stXStage.bLimitForwardEnable := TRUE;
stXStage.bLimitBackwardEnable := TRUE;
stXStage.bHardwareEnable := TRUE;
stXStage.bPowerSelf := TRUE;

fbYStage(stMotionStage:=stYStage);
fbXStage(stMotionStage:=stXStage);

// We need to update from PLC or from EPICS, but not both
fbArrCheckWrite(
    astPositionState:=astPositionState,
    bCheck:=TRUE,
    bSave:=FALSE,
);
IF NOT fbArrCheckWrite.bHadWrite THEN
    astPositionState[ENUM_TM2K4_States.OUT] := stOut;
    astPositionState[ENUM_TM2K4_States.TARGET1a] := stTarget1a;
    astPositionState[ENUM_TM2K4_States.TARGET1b] := stTarget1b;
    astPositionState[ENUM_TM2K4_States.TARGET2a] := stTarget2a;
    astPositionState[ENUM_TM2K4_States.TARGET2b] := stTarget2b;
    astPositionState[ENUM_TM2K4_States.TARGET3a] := stTarget3a;
    astPositionState[ENUM_TM2K4_States.TARGET3b] := stTarget3b;
    astPositionState[ENUM_TM2K4_States.YAG] := stTarget4;
    astPositionState[ENUM_TM2K4_States.DIODE] := stTarget5;
END_IF

fbStates(
    stMotionStage:=stYStage,
    astPositionState:=astPositionState,
    eEnumSet:=eEnumSet,
    eEnumGet:=eEnumGet,
    fbFFHWO:=fbFFHWO,
    fbArbiter:=fbArbiter,
    bEnableMotion:=bEnableMotion,
    bEnableBeamParams:=bEnableBeamParams,
    bEnablePositionLimits:=bEnablePositionLimits,
    sDeviceName:=sDeviceName,
    sTransitionKey:=sTransitionKey,
    bReadDBNow:=bReadDBNow,
    stDbStateParams=>stDbStateParams,
);

fbArrCheckWrite(
    astPositionState:=astPositionState,
    bCheck:=FALSE,
    bSave:=TRUE,
);

stOut := astPositionState[ENUM_TM2K4_States.OUT];
stTarget1a := astPositionState[ENUM_TM2K4_States.TARGET1a];
stTarget1b := astPositionState[ENUM_TM2K4_States.TARGET1b];
stTarget2a := astPositionState[ENUM_TM2K4_States.TARGET2a];
stTarget2b := astPositionState[ENUM_TM2K4_States.TARGET2b];
stTarget3a := astPositionState[ENUM_TM2K4_States.TARGET3a];
stTarget3b := astPositionState[ENUM_TM2K4_States.TARGET3b];
stTarget4 := astPositionState[ENUM_TM2K4_States.YAG];
stTarget5 := astPositionState[ENUM_TM2K4_States.DIODE];

fbTempSensor1(
    fFaultThreshold:=fbStates.stDbStateParams.stReactiveParams.nTempSP,
    bVeto:=eEnumGet = ENUM_TM2K4_States.OUT,
    sDevName:=sDeviceName,
    io_fbFFHWO:=fbFFHWO,
);
fbFlowMeter();

END_FUNCTION_BLOCK

// ---- POUs/PRG_SP1K4.TcPOU
  PROGRAM PRG_SP1K4
VAR
    fbMotionLensX: FB_MotionStage;
    fbMotionFoilX: FB_MotionStage;
    fbMotionZPX: FB_MotionStage;
    fbMotionZPY: FB_MotionStage;
    fbMotionZPZ: FB_MotionStage;
    fbMotionYAGX: FB_MotionStage;
    fbMotionYAGY: FB_MotionStage;
    fbMotionYAGZ: FB_MotionStage;
    fbMotionYAGR: FB_MotionStage;
    fbMotionTL1: FB_MotionStage;
    fbMotionTL2: FB_MotionStage;
    fbMotionTLX: FB_MotionStage;
    fbMotionFoilY: FB_MotionStage;

    {attribute 'TcLinkTo' := 'TIIB[LensX_EL1004]^Channel 1^Input'}
    bHallInput1 AT %I* : BOOL;

    {attribute 'TcLinkTo' := 'TIIB[LensX_EL1004]^Channel 2^Input'}
    bHallInput2 AT %I* : BOOL;

    {attribute 'TcLinkTo' := 'TIIB[SP1K4-TL1-EL1124]^Channel 1^Input'}
    bTL1High AT %I*: BOOL;
    nTL1HighCycles: UINT;
    {attribute 'TcLinkTo' := 'TIIB[SP1K4-TL1-EL1124]^Channel 2^Input'}
    bTL1Low AT %I*: BOOL;
    nTL1LowCycles: UINT;
    {attribute 'TcLinkTo' := 'TIIB[SP1K4-TL2-EL1124]^Channel 1^Input'}
    bTL2High AT %I*: BOOL;
    nTL2HighCycles: UINT;
    {attribute 'TcLinkTo' := 'TIIB[SP1K4-TL2-EL1124]^Channel 2^Input'}
    bTL2Low AT %I*: BOOL;
    nTL2LowCycles: UINT;

    nNumCyclesNeeded: UINT := 100;

    bInit: BOOL :=TRUE;

    // Placeholder, later this should be TRUE if the attenuator is in and FALSE otherwise
    bAttIn: BOOL;

    ////ZP states start
    {attribute 'pytmc' := '
        pv: SP1K4:FZP
    '}
    fbZPStates: FB_PositionStatePMPS3D;
    {attribute 'pytmc' := '
        pv: SP1K4:FZP:STATE:SET
        io: io
    '}
    zp_enumSet: ENUM_ZonePlate_States;
     {attribute 'pytmc' := '
        pv: SP1K4:FZP:STATE:GET
        io: io
    '}
    zp_enumGet: ENUM_ZonePlate_States;
    fbZPSetup: FB_StateSetupHelper;
    fbZPDefault: ST_PositionState := (
        fDelta:=1.5,
        fVelocity:=3.0,
 //       bMoveOk:=TRUE,
        bValid:=TRUE
    );
    aZPXStates: ARRAY[1..GeneralConstants.MAX_STATES] OF ST_PositionState;
    aZPYStates: ARRAY[1..GeneralConstants.MAX_STATES] OF ST_PositionState;
    aZPZStates: ARRAY[1..GeneralConstants.MAX_STATES] OF ST_PositionState;

    ////Solid-ATT states start
    {attribute 'pytmc' := '
        pv: SP1K4:ATT
    '}
    fbATTStates: FB_PositionStatePMPS2D;
    {attribute 'pytmc' := '
        pv: SP1K4:ATT:STATE:SET
        io: io
    '}
    att_enumSet: ENUM_SolidAttenuator_States;
     {attribute 'pytmc' := '
        pv: SP1K4:ATT:STATE:GET
        io: i
    '}
    att_enumGet: ENUM_SolidAttenuator_States;
    fbATTSetup: FB_StateSetupHelper;
    fbATTDefault: ST_PositionState := (
        fDelta:=2.0,
        fVelocity:=2,
//        bMoveOk:=TRUE,
        bValid:=TRUE
    );
    aATTXStates: ARRAY[1..GeneralConstants.MAX_STATES] OF ST_PositionState;
    aATTYStates: ARRAY[1..GeneralConstants.MAX_STATES] OF ST_PositionState;

    bPF1K4Out: BOOL;

    // SP1K4 RTD-01
    {attribute 'TcLinkTo' := '.iRaw := TIIB[SP1K4-EL3202-E9A]^RTD Inputs Channel 1^Value;
                              .bUnderrange := TIIB[SP1K4-EL3202-E9A]^RTD Inputs Channel 1^Status^Underrange;
                              .bOverrange := TIIB[SP1K4-EL3202-E9A]^RTD Inputs Channel 1^Status^Overrange;
                              .bError := TIIB[SP1K4-EL3202-E9A]^RTD Inputs Channel 1^Status^Error'}
    {attribute 'pytmc' := '
        pv: TMO:SPEC:RTD:01
        field: EGU C
        io: i
    '}
    SP1K4_ATT_RTD_01 : FB_CC_TempSensor;

    {attribute 'TcLinkTo' := '.iRaw := TIIB[SP1K4-EL3202-E9A]^RTD Inputs Channel 2^Value;
                              .bUnderrange := TIIB[SP1K4-EL3202-E9A]^RTD Inputs Channel 2^Status^Underrange;
                              .bOverrange := TIIB[SP1K4-EL3202-E9A]^RTD Inputs Channel 2^Status^Overrange;
                              .bError := TIIB[SP1K4-EL3202-E9A]^RTD Inputs Channel 2^Status^Error'}
    {attribute 'pytmc' := '
        pv: TMO:SPEC:RTD:02
        field: EGU C
        io: i
    '}
    SP1K4_ATT_RTD_02 : FB_CC_TempSensor;

    {attribute 'TcLinkTo' := '.iRaw := TIIB[EP3174-FWM-E2]^AI Standard Channel 2^Value'}
    {attribute 'pytmc' :='pv: TMO:SPEC'}
    fbFlowMeter: FB_FDQ_FlowMeter;
END_VAR

 bPF1K4Out := GVL_TcGVL.ePF1K4State = E_WFS_States.OUT;
// Hardware Enable and fbMotionStage
//Lens X
Main.M32.bLimitForwardEnable := NOT bHallInput1;
Main.M32.bLimitBackwardEnable := NOT bHallInput2;
fbMotionLensX(stMotionStage:=Main.M32);


//Zone Plate
fbMotionZPX(stMotionStage:=Main.M34);
fbMotionZPY(stMotionStage:=Main.M35);
fbMotionZPZ(stMotionStage:=Main.M36);

fbZPSetup(stPositionState:=fbZPDefault, bSetDefault:=TRUE);
//swap several FZP targets for run 24 3-18-25
fbZPSetup(stPositionState:=aZPXStates[ENUM_ZonePlate_States.OUT], sName:='OUT', fPosition:=15);
fbZPSetup(stPositionState:=aZPYStates[ENUM_ZonePlate_States.OUT], sName:='OUT', fPosition:=-3.5);
fbZPSetup(stPositionState:=aZPZStates[ENUM_ZonePlate_States.OUT], sName:='OUT', fPosition:=0);

fbZPSetup(stPositionState:=aZPXStates[ENUM_ZonePlate_States.Target1b], sName:='YAG', fPosition:=49);
fbZPSetup(stPositionState:=aZPYStates[ENUM_ZonePlate_States.Target1b], sName:='YAG', fPosition:=0.65);
fbZPSetup(stPositionState:=aZPZStates[ENUM_ZonePlate_States.Target1b], sName:='YAG', fPosition:=0);

//paddle3
fbZPSetup(stPositionState:=aZPXStates[ENUM_ZonePlate_States.Target5a], sName:='FZP-260_1', fPosition:=81);
fbZPSetup(stPositionState:=aZPYStates[ENUM_ZonePlate_States.Target5a], sName:='FZP-260_1', fPosition:=-8.2);
fbZPSetup(stPositionState:=aZPZStates[ENUM_ZonePlate_States.Target5a], sName:='FZP-260_1', fPosition:=0);

fbZPSetup(stPositionState:=aZPXStates[ENUM_ZonePlate_States.Target4b], sName:='FZP-1212_1', fPosition:=73);
fbZPSetup(stPositionState:=aZPYStates[ENUM_ZonePlate_States.Target4b], sName:='FZP-1212_1', fPosition:=0.65);
fbZPSetup(stPositionState:=aZPZStates[ENUM_ZonePlate_States.Target4b], sName:='FZP-1212_1', fPosition:=0);

fbZPSetup(stPositionState:=aZPXStates[ENUM_ZonePlate_States.Target5b], sName:='FZP-350_1', fPosition:=81);
fbZPSetup(stPositionState:=aZPYStates[ENUM_ZonePlate_States.Target5b], sName:='FZP-350_1', fPosition:=0.65);
fbZPSetup(stPositionState:=aZPZStates[ENUM_ZonePlate_States.Target5b], sName:='FZP-350_1', fPosition:=0);
//paddle is changed on 4-30-25
fbZPSetup(stPositionState:=aZPXStates[ENUM_ZonePlate_States.Target3b], sName:='FZP-806_1', fPosition:=65);
fbZPSetup(stPositionState:=aZPYStates[ENUM_ZonePlate_States.Target3b], sName:='FZP-806_1', fPosition:=0.65);
fbZPSetup(stPositionState:=aZPZStates[ENUM_ZonePlate_States.Target3b], sName:='FZP-806_1', fPosition:=0);
//paddle is changed on 4-30-25
fbZPSetup(stPositionState:=aZPXStates[ENUM_ZonePlate_States.Target2b], sName:='FZP-690_1', fPosition:=57);
fbZPSetup(stPositionState:=aZPYStates[ENUM_ZonePlate_States.Target2b], sName:='FZP-690_1', fPosition:=0.65);
fbZPSetup(stPositionState:=aZPZStates[ENUM_ZonePlate_States.Target2b], sName:='FZP-690_1', fPosition:=0);

fbZPSetup(stPositionState:=aZPXStates[ENUM_ZonePlate_States.Target1a], sName:='FZP-530_1', fPosition:=49);
fbZPSetup(stPositionState:=aZPYStates[ENUM_ZonePlate_States.Target1a], sName:='FZP-530_1', fPosition:=-8.2);
fbZPSetup(stPositionState:=aZPZStates[ENUM_ZonePlate_States.Target1a], sName:='FZP-530_1', fPosition:=0);

fbZPSetup(stPositionState:=aZPXStates[ENUM_ZonePlate_States.Target2a], sName:='FZP-530_2', fPosition:=57);
fbZPSetup(stPositionState:=aZPYStates[ENUM_ZonePlate_States.Target2a], sName:='FZP-530_2', fPosition:=-8.2);
fbZPSetup(stPositionState:=aZPZStates[ENUM_ZonePlate_States.Target2a], sName:='FZP-530_2', fPosition:=0);
// FZP-690-1 position X and Y are chanegd due to last TMO MRCO shift 3-7-2025
fbZPSetup(stPositionState:=aZPXStates[ENUM_ZonePlate_States.Target6b], sName:='FZP-262-524-dual_1', fPosition:=88.882);
fbZPSetup(stPositionState:=aZPYStates[ENUM_ZonePlate_States.Target6b], sName:='FZP-262-524-dual_1', fPosition:=-0.0144);
fbZPSetup(stPositionState:=aZPZStates[ENUM_ZonePlate_States.Target6b], sName:='FZP-262-524-dual_1', fPosition:=0);

fbZPSetup(stPositionState:=aZPXStates[ENUM_ZonePlate_States.Target7b], sName:='FZP-262-524-dual_2', fPosition:=97);
fbZPSetup(stPositionState:=aZPYStates[ENUM_ZonePlate_States.Target7b], sName:='FZP-262-524-dual_2', fPosition:=0.5);
fbZPSetup(stPositionState:=aZPZStates[ENUM_ZonePlate_States.Target7b], sName:='FZP-262-524-dual_2', fPosition:=0);

fbZPSetup(stPositionState:=aZPXStates[ENUM_ZonePlate_States.Target6a], sName:='FZP-400_1', fPosition:=89);
fbZPSetup(stPositionState:=aZPYStates[ENUM_ZonePlate_States.Target6a], sName:='FZP-400_1', fPosition:=-8.2);
fbZPSetup(stPositionState:=aZPZStates[ENUM_ZonePlate_States.Target6a], sName:='FZP-400_1', fPosition:=0);

fbZPSetup(stPositionState:=aZPXStates[ENUM_ZonePlate_States.Target7a], sName:='FZP-400_2', fPosition:=97);
fbZPSetup(stPositionState:=aZPYStates[ENUM_ZonePlate_States.Target7a], sName:='FZP-400_2', fPosition:=-8.2);
fbZPSetup(stPositionState:=aZPZStates[ENUM_ZonePlate_States.Target7a], sName:='FZP-400_2', fPosition:=0);

fbZPSetup(stPositionState:=aZPXStates[ENUM_ZonePlate_States.Target3a], sName:='FZP-613.5_1', fPosition:=65);
fbZPSetup(stPositionState:=aZPYStates[ENUM_ZonePlate_States.Target3a], sName:='FZP-613.5_1', fPosition:=-8.2);
fbZPSetup(stPositionState:=aZPZStates[ENUM_ZonePlate_States.Target3a], sName:='FZP-613.5_1', fPosition:=0);

fbZPSetup(stPositionState:=aZPXStates[ENUM_ZonePlate_States.Target4a], sName:='FZP-613.5_2', fPosition:=73);
fbZPSetup(stPositionState:=aZPYStates[ENUM_ZonePlate_States.Target4a], sName:='FZP-613.5_2', fPosition:=-8.2);
fbZPSetup(stPositionState:=aZPZStates[ENUM_ZonePlate_States.Target4a], sName:='FZP-613.5_2', fPosition:=0);


//paddle3
aZPXStates[ENUM_ZonePlate_States.OUT].bMoveOk := TRUE;
aZPXStates[ENUM_ZonePlate_States.Target1b].bMoveOk := bPF1K4Out;
aZPXStates[ENUM_ZonePlate_States.Target5a].bMoveOK := bPF1K4Out;
aZPXStates[ENUM_ZonePlate_States.Target4b].bMoveOK := bPF1K4Out;
aZPXStates[ENUM_ZonePlate_States.Target5b].bMoveOK := bPF1K4Out;
aZPXStates[ENUM_ZonePlate_States.Target3b].bMoveOK := bPF1K4Out;
aZPXStates[ENUM_ZonePlate_States.Target2b].bMoveOK := bPF1K4Out;
aZPXStates[ENUM_ZonePlate_States.Target1a].bMoveOK := bPF1K4Out;
aZPXStates[ENUM_ZonePlate_States.Target2a].bMoveOK := bPF1K4Out;
aZPXStates[ENUM_ZonePlate_States.Target6b].bMoveOK := bPF1K4Out;
aZPXStates[ENUM_ZonePlate_States.Target7b].bMoveOK := bPF1K4Out;
aZPXStates[ENUM_ZonePlate_States.Target6a].bMoveOK := bPF1K4Out;
aZPXStates[ENUM_ZonePlate_States.Target7a].bMoveOK := bPF1K4Out;
aZPXStates[ENUM_ZonePlate_States.Target3a].bMoveOK := bPF1K4Out;
aZPXStates[ENUM_ZonePlate_States.Target4a].bMoveOK := bPF1K4Out;

aZPYStates[ENUM_ZonePlate_States.OUT].bMoveOk := TRUE;
aZPYStates[ENUM_ZonePlate_States.Target1b].bMoveOk := bPF1K4Out;
aZPYStates[ENUM_ZonePlate_States.Target5a].bMoveOK := bPF1K4Out;
aZPYStates[ENUM_ZonePlate_States.Target4b].bMoveOK := bPF1K4Out;
aZPYStates[ENUM_ZonePlate_States.Target5b].bMoveOK := bPF1K4Out;
aZPYStates[ENUM_ZonePlate_States.Target3b].bMoveOK := bPF1K4Out;
aZPYStates[ENUM_ZonePlate_States.Target2b].bMoveOK := bPF1K4Out;
aZPYStates[ENUM_ZonePlate_States.Target1a].bMoveOK := bPF1K4Out;
aZPYStates[ENUM_ZonePlate_States.Target2a].bMoveOK := bPF1K4Out;
aZPYStates[ENUM_ZonePlate_States.Target6b].bMoveOK := bPF1K4Out;
aZPYStates[ENUM_ZonePlate_States.Target7b].bMoveOK := bPF1K4Out;
aZPYStates[ENUM_ZonePlate_States.Target6a].bMoveOK := bPF1K4Out;
aZPYStates[ENUM_ZonePlate_States.Target7a].bMoveOK := bPF1K4Out;
aZPYStates[ENUM_ZonePlate_States.Target3a].bMoveOK := bPF1K4Out;
aZPYStates[ENUM_ZonePlate_States.Target4a].bMoveOK := bPF1K4Out;

aZPZStates[ENUM_ZonePlate_States.OUT].bMoveOk := TRUE;
aZPZStates[ENUM_ZonePlate_States.Target1b].bMoveOk := bPF1K4Out;
aZPZStates[ENUM_ZonePlate_States.Target5a].bMoveOK := bPF1K4Out;
aZPZStates[ENUM_ZonePlate_States.Target4b].bMoveOK := bPF1K4Out;
aZPZStates[ENUM_ZonePlate_States.Target5b].bMoveOK := bPF1K4Out;
aZPZStates[ENUM_ZonePlate_States.Target3b].bMoveOK := bPF1K4Out;
aZPZStates[ENUM_ZonePlate_States.Target2b].bMoveOK := bPF1K4Out;
aZPZStates[ENUM_ZonePlate_States.Target1a].bMoveOK := bPF1K4Out;
aZPZStates[ENUM_ZonePlate_States.Target2a].bMoveOK := bPF1K4Out;
aZPZStates[ENUM_ZonePlate_States.Target6b].bMoveOK := bPF1K4Out;
aZPZStates[ENUM_ZonePlate_States.Target7b].bMoveOK := bPF1K4Out;
aZPZStates[ENUM_ZonePlate_States.Target6a].bMoveOK := bPF1K4Out;
aZPZStates[ENUM_ZonePlate_States.Target7a].bMoveOK := bPF1K4Out;
aZPZStates[ENUM_ZonePlate_States.Target3a].bMoveOK := bPF1K4Out;
aZPZStates[ENUM_ZonePlate_States.Target4a].bMoveOK := bPF1K4Out;

bAttIn := att_enumGet <> ENUM_SolidAttenuator_States.OUT AND  att_enumGet <> ENUM_SolidAttenuator_States.Unknown;


//paddle2
IF bAttIn THEN
    // Attenuator is in, pick the ATT_IN states
    aZPXStates[ENUM_ZonePlate_States.OUT].stPMPS.sPmpsState := 'SP1K4:FZP-OUT';
    aZPXStates[ENUM_ZonePlate_States.Target1b].stPMPS.sPmpsState := 'SP1K4:FZP-Target1b_ATT_IN';
    aZPXStates[ENUM_ZonePlate_States.Target5a].stPMPS.sPmpsState := 'SP1K4:FZP-Target5a_ATT_IN';
    aZPXStates[ENUM_ZonePlate_States.Target4b].stPMPS.sPmpsState := 'SP1K4:FZP-Target4b_ATT_IN';
    aZPXStates[ENUM_ZonePlate_States.Target5b].stPMPS.sPmpsState := 'SP1K4:FZP-Target5b_ATT_IN';
    aZPXStates[ENUM_ZonePlate_States.Target3b].stPMPS.sPmpsState := 'SP1K4:FZP-Target3b_ATT_IN';
    aZPXStates[ENUM_ZonePlate_States.Target2b].stPMPS.sPmpsState := 'SP1K4:FZP-Target2b_ATT_IN';
    aZPXStates[ENUM_ZonePlate_States.Target1a].stPMPS.sPmpsState := 'SP1K4:FZP-Target1a_ATT_IN';
    aZPXStates[ENUM_ZonePlate_States.Target2a].stPMPS.sPmpsState := 'SP1K4:FZP-Target2a_ATT_IN';
    aZPXStates[ENUM_ZonePlate_States.Target6b].stPMPS.sPmpsState := 'SP1K4:FZP-Target6b_ATT_IN';
    aZPXStates[ENUM_ZonePlate_States.Target7b].stPMPS.sPmpsState := 'SP1K4:FZP-Target7b_ATT_IN';
    aZPXStates[ENUM_ZonePlate_States.Target6a].stPMPS.sPmpsState := 'SP1K4:FZP-Target6a_ATT_IN';
    aZPXStates[ENUM_ZonePlate_States.Target7a].stPMPS.sPmpsState := 'SP1K4:FZP-Target7a_ATT_IN';
    aZPXStates[ENUM_ZonePlate_States.Target3a].stPMPS.sPmpsState := 'SP1K4:FZP-Target3a_ATT_IN';
    aZPXStates[ENUM_ZonePlate_States.Target4a].stPMPS.sPmpsState := 'SP1K4:FZP-Target4a_ATT_IN';

ELSE
    // Attenuator is out, pick the ATT_OUT states
    aZPXStates[ENUM_ZonePlate_States.OUT].stPMPS.sPmpsState := 'SP1K4:FZP-OUT';
    aZPXStates[ENUM_ZonePlate_States.Target1b].stPMPS.sPmpsState := 'SP1K4:FZP-Target1b_ATT_OUT';
    aZPXStates[ENUM_ZonePlate_States.Target5a].stPMPS.sPmpsState := 'SP1K4:FZP-Target5a_ATT_OUT';
    aZPXStates[ENUM_ZonePlate_States.Target4b].stPMPS.sPmpsState := 'SP1K4:FZP-Target4b_ATT_OUT';
    aZPXStates[ENUM_ZonePlate_States.Target5b].stPMPS.sPmpsState := 'SP1K4:FZP-Target5b_ATT_OUT';
    aZPXStates[ENUM_ZonePlate_States.Target3b].stPMPS.sPmpsState := 'SP1K4:FZP-Target3b_ATT_OUT';
    aZPXStates[ENUM_ZonePlate_States.Target2b].stPMPS.sPmpsState := 'SP1K4:FZP-Target2b_ATT_OUT';
    aZPXStates[ENUM_ZonePlate_States.Target1a].stPMPS.sPmpsState := 'SP1K4:FZP-Target1a_ATT_OUT';
    aZPXStates[ENUM_ZonePlate_States.Target2a].stPMPS.sPmpsState := 'SP1K4:FZP-Target2a_ATT_OUT';
    aZPXStates[ENUM_ZonePlate_States.Target6b].stPMPS.sPmpsState := 'SP1K4:FZP-Target6b_ATT_OUT';
    aZPXStates[ENUM_ZonePlate_States.Target7b].stPMPS.sPmpsState := 'SP1K4:FZP-Target7b_ATT_OUT';
    aZPXStates[ENUM_ZonePlate_States.Target6a].stPMPS.sPmpsState := 'SP1K4:FZP-Target6a_ATT_OUT';
    aZPXStates[ENUM_ZonePlate_States.Target7a].stPMPS.sPmpsState := 'SP1K4:FZP-Target7a_ATT_OUT';
    aZPXStates[ENUM_ZonePlate_States.Target3a].stPMPS.sPmpsState := 'SP1K4:FZP-Target3a_ATT_OUT';
    aZPXStates[ENUM_ZonePlate_States.Target4a].stPMPS.sPmpsState := 'SP1K4:FZP-Target4a_ATT_OUT';
END_IF

fbZPStates(
    stMotionStage1:=Main.M34,
    stMotionStage2:=Main.M35,
    stMotionStage3:=Main.M36,
    astPositionState1:=aZPXStates,
    astPositionState2:=aZPYStates,
    astPositionState3:=aZPZStates,
    eEnumSet:=zp_enumSet,
    eEnumGet:=zp_enumGet,
    fbFFHWO:=fbFastFaultOutput1,
    fbArbiter:=fbArbiter,
    bEnableMotion:=TRUE,
    bEnableBeamParams:=TRUE,
    bEnablePositionLimits:=TRUE,
    sDeviceName:='SP1K4:FZP',
    sTransitionKey:='SP1K4:FZP-TRANSITION',
);


// Foil X (Solid-ATT-X)
fbMotionFoilX(stMotionStage:=Main.M33);


// YAG
fbMotionYAGX(stMotionStage:=Main.M37);
fbMotionYAGY(stMotionStage:=Main.M38);
fbMotionYAGZ(stMotionStage:=Main.M39);
fbMotionYAGR(stMotionStage:=Main.M40);
// Thorlabs
fbMotionTL1(stMotionStage:=Main.M41);
fbMotionTL2(stMotionStage:=Main.M42);
//Thorlab-LenX
fbMotionTLX(stMotionStage:=Main.M43);
//FOIL Y (Solid-ATT-Y)
fbMotionFoilY(stMotionStage:=Main.M44);




// SP1K4-SOLID-ATT PMPS
fbATTSetup(stPositionState:=fbATTDefault, bSetDefault:=TRUE);

fbATTSetup(stPositionState:=aATTXStates[ENUM_SolidAttenuator_States.OUT], sName:='OUT', fPosition:=11.0);
fbATTSetup(stPositionState:=aATTYStates[ENUM_SolidAttenuator_States.OUT], sName:='OUT', fPosition:=1.00);

fbATTSetup(stPositionState:=aATTXStates[ENUM_SolidAttenuator_States.Target1], sName:='TARGET1', fPosition:=36.5625);
fbATTSetup(stPositionState:=aATTYStates[ENUM_SolidAttenuator_States.Target1], sName:='TARGET1', fPosition:=2.2);

fbATTSetup(stPositionState:=aATTXStates[ENUM_SolidAttenuator_States.Target2], sName:='TARGET2', fPosition:=54.5);
fbATTSetup(stPositionState:=aATTYStates[ENUM_SolidAttenuator_States.Target2], sName:='TARGET2', fPosition:=2.0);

fbATTSetup(stPositionState:=aATTXStates[ENUM_SolidAttenuator_States.Target3], sName:='TARGET3', fPosition:=72.2);
fbATTSetup(stPositionState:=aATTYStates[ENUM_SolidAttenuator_States.Target3], sName:='TARGET3', fPosition:=1.6);

fbATTSetup(stPositionState:=aATTXStates[ENUM_SolidAttenuator_States.Target4], sName:='TARGET4', fPosition:=90.2);
fbATTSetup(stPositionState:=aATTYStates[ENUM_SolidAttenuator_States.Target4], sName:='TARGET4', fPosition:=1.3);

fbATTSetup(stPositionState:=aATTXStates[ENUM_SolidAttenuator_States.Target5], sName:='TARGET5', fPosition:=107.8);
fbATTSetup(stPositionState:=aATTYStates[ENUM_SolidAttenuator_States.Target5], sName:='TARGET5', fPosition:=1.0);

aATTXStates[ENUM_SolidAttenuator_States.OUT].bMoveOk := TRUE;
aATTXStates[ENUM_SolidAttenuator_States.Target1].bMoveOk := bPF1K4Out;
aATTXStates[ENUM_SolidAttenuator_States.Target2].bMoveOk := bPF1K4Out;
aATTXStates[ENUM_SolidAttenuator_States.Target3].bMoveOk := bPF1K4Out;
aATTXStates[ENUM_SolidAttenuator_States.Target4].bMoveOk := bPF1K4Out;
aATTXStates[ENUM_SolidAttenuator_States.Target5].bMoveOk := bPF1K4Out;


aATTYStates[ENUM_SolidAttenuator_States.OUT].bMoveOk := TRUE;
aATTYStates[ENUM_SolidAttenuator_States.Target1].bMoveOk := bPF1K4Out;
aATTYStates[ENUM_SolidAttenuator_States.Target2].bMoveOk := bPF1K4Out;
aATTYStates[ENUM_SolidAttenuator_States.Target3].bMoveOk := bPF1K4Out;
aATTYStates[ENUM_SolidAttenuator_States.Target4].bMoveOk := bPF1K4Out;
aATTYStates[ENUM_SolidAttenuator_States.Target5].bMoveOk := bPF1K4Out;





aATTXStates[ENUM_SolidAttenuator_States.OUT].stPMPS.sPmpsState := 'SP1K4:ATT-OUT';
aATTXStates[ENUM_SolidAttenuator_States.Target1].stPMPS.sPmpsState := 'SP1K4:ATT-TARGET1';
aATTXStates[ENUM_SolidAttenuator_States.Target2].stPMPS.sPmpsState := 'SP1K4:ATT-TARGET2';
aATTXStates[ENUM_SolidAttenuator_States.Target3].stPMPS.sPmpsState := 'SP1K4:ATT-TARGET3';
aATTXStates[ENUM_SolidAttenuator_States.Target4].stPMPS.sPmpsState := 'SP1K4:ATT-TARGET4';
aATTXStates[ENUM_SolidAttenuator_States.Target5].stPMPS.sPmpsState := 'SP1K4:ATT-TARGET5';

fbATTStates(
    stMotionStage1:=Main.M33,
    stMotionStage2:=Main.M44,
    astPositionState1:=aATTXStates,
    astPositionState2:=aATTYStates,
    eEnumSet:=att_enumSet,
    eEnumGet:=att_enumGet,
    fbFFHWO:=fbFastFaultOutput1,
    fbArbiter:=fbArbiter,
    bEnableMotion:=TRUE,
    bEnableBeamParams:=TRUE,
    bEnablePositionLimits:=TRUE,
    sDeviceName:='SP1K4:ATT',
    sTransitionKey:='SP1K4:ATT-TRANSITION',
);








IF NOT bTL1High THEN
    nTL1HighCycles := MIN(nTL1HighCycles + 1, nNumCyclesNeeded);
ELSE
    nTL1HighCycles := 0;
END_IF
IF NOT bTL1Low THEN
    nTL1LowCycles := MIN(nTL1LowCycles + 1, nNumCyclesNeeded);
ELSE
    nTL1LowCycles := 0;
END_IF
IF NOT bTL2High THEN
    nTL2HighCycles := MIN(nTL2HighCycles + 1, nNumCyclesNeeded);
ELSE
    nTL2HighCycles := 0;
END_IF
IF NOT bTL2Low THEN
    nTL2LowCycles := MIN(nTL2LowCycles + 1, nNumCyclesNeeded);
ELSE
    nTL2LowCycles := 0;
END_IF

Main.M41.bLimitForwardEnable := nTL1HighCycles < nNumCyclesNeeded;
Main.M41.bLimitBackwardEnable := nTL1LowCycles < nNumCyclesNeeded;
Main.M42.bLimitForwardEnable := nTL2HighCycles < nNumCyclesNeeded;
Main.M42.bLimitBackwardEnable := nTL2LowCycles < nNumCyclesNeeded;
Main.M43.bLimitBackwardEnable := True;
Main.M43.bLimitForwardEnable := True;

GVL_TcGVL.eSP1K4FZP := zp_enumGet;
GVL_TcGVL.eSP1K4ATT := att_enumGet;

SP1K4_ATT_RTD_01(
    fResolution:=0.01,
    fFaultThreshold:=fbAttStates.stDbStateParams.stReactiveParams.nTempSP,
    bVeto:=att_enumGet = ENUM_SolidAttenuator_States.OUT,
    sDevName:='SP1K4:ATT',
    io_fbFFHWO:=fbFastFaultOutput1,

);
SP1K4_ATT_RTD_02(
    fResolution:=0.01,
    fFaultThreshold:=fbAttStates.stDbStateParams.stReactiveParams.nTempSP,
    bVeto:=att_enumGet = ENUM_SolidAttenuator_States.OUT,
    sDevName:='SP1K4:ATT',
    io_fbFFHWO:=fbFastFaultOutput1,
);

fbFlowMeter();

END_PROGRAM

// ---- POUs/PRG_LI2K4_IP1.TcPOU
PROGRAM PRG_LI2K4_IP1
VAR

    fbMotionLI2K4X: FB_MotionStage;
    fbMotionLI2K4Y: FB_MotionStage;

    bLI2K4StatesReset : BOOL;
    anStateSequenceOrderLI2K4Y : ARRAY[1...GeneralConstants.MAX_STATES] OF UINT;
    anStateSequenceOrderLI2K4X : ARRAY[1...GeneralConstants.MAX_STATES] OF UINT;
    fbLI2K4YStates: FB_PositionStatePMPS1D;
    fbLI2K4XStates: FB_PositionStatePMPS1D;
    fbFastFault: FB_FastFault;

    {attribute 'pytmc' := '
        pv: LI2K4:IP1
        io: io
    '}
    fbLI2K4States : FB_SequenceMover2D;
    //fbLI2K4States : FB_PositionStatePMPS2D;

    {attribute 'pytmc' := '
        pv: LI2K4:IP1:STATE:SET
        io: io
    '}
    li2k4_enumSet: ENUM_LaserCoupling_States;
     {attribute 'pytmc' := '
        pv: LI2K4:IP1:STATE:GET
        io: i
    '}
    li2k4_enumGet: ENUM_LaserCoupling_States;
    fbStateSetup: FB_StateSetupHelper;
    stDefault: ST_PositionState :=(
  //      fDelta :=0.5,
        fVelocity := 2.0,
        bMoveOk := TRUE,
        bValid := TRUE
    );
    aLI2K4XStates: ARRAY[1..GeneralConstants.MAX_STATES] OF ST_PositionState;
    aLI2K4YStates: ARRAY[1..GeneralConstants.MAX_STATES] OF ST_PositionState;

    EPS_LI2K4Y_Positive : FB_EPS;
    EPS_LI2K4Y_Negative : FB_EPS;
    EPS_LI2K4X_Positive : FB_EPS;
    EPS_LI2K4X_Negative : FB_EPS;
END_VAR

//IF Main.M46.stAxisStatus.fActPosition < -0.85 THEN
//   Main.M45.fVelocity := 0.01;
//END_IF
//IF Main.M45.stAxisStatus.fActPosition > 85 THEN
//   Main.M46.bExecute := FALSE;
//END_IF

fbMotionLI2K4Y(stMotionStage:=Main.M45);
fbMotionLI2K4X(stMotionStage:=Main.M46);

//LI2K4 2DPMPS
fbStateSetup(stPositionState:=stDefault, bSetDefault:=TRUE);
fbStateSetup(stPositionState:=aLI2K4XStates[ENUM_LaserCoupling_States.OUT], fDelta := 0.1, sName := 'OUT', fPosition:=-0.214);

fbStateSetup(stPositionState:=aLI2K4YStates[ENUM_LaserCoupling_States.OUT], fDelta := 0.5,  sName := 'OUT', fPosition:=133.0);
fbStateSetup(stPositionState:=aLI2K4XStates[ENUM_LaserCoupling_States.Mirror1],fDelta := 0.4, sName := 'MIRROR1', fPosition:=-0.795);
fbStateSetup(stPositionState:=aLI2K4YStates[ENUM_LaserCoupling_States.Mirror1],fDelta := 0.5, sName := 'MIRROR1', fPosition:=80.896);

aLI2K4YStates[ENUM_LaserCoupling_States.OUT].stPMPS.sPmpsState := 'LI2K4:IP1-OUT';
aLI2K4YStates[ENUM_LaserCoupling_States.Mirror1].stPMPS.sPmpsState := 'LI2K4:IP1-MIRROR1';
aLI2K4XStates[ENUM_LaserCoupling_States.OUT].stPMPS.sPmpsState := 'LI2K4:IP1-OUT';
aLI2K4XStates[ENUM_LaserCoupling_States.Mirror1].stPMPS.sPmpsState := 'LI2K4:IP1-MIRROR1';

(* The LI2K4 sequence mover is insteded to move as follows:
   When moving from OUT to MIRROR1, first Y is moved, then once Y movement is complete, X is moved.
When moving from MIRROR1 to OUT, first X is moved, then once X movement is complete, Y is moved.
*)
EPS_LI2K4Y_Positive(eps:=Main.M45.stEPSForwardEnable);
EPS_LI2K4Y_Positive.setBit(nBits := 0, bValue:= Main.M46.stAxisStatus.fActPosition > -0.3 OR Main.M45.stAxisStatus.fActPosition < 82);
EPS_LI2K4Y_Negative(eps:=Main.M45.stEPSBackwardEnable);
EPS_LI2K4Y_Negative.setBit(nBits := 0, bValue:= Main.M46.stAxisStatus.fActPosition > -0.3 OR Main.M45.stAxisStatus.fActPosition > 79);

EPS_LI2K4X_Positive(eps:=Main.M46.stEPSForwardEnable);
EPS_LI2K4X_Positive.setBit(nBits := 0, bValue:= Main.M45.stAxisStatus.fActPosition < 82 OR Main.M46.stAxisStatus.fActPosition < -0.114);
EPS_LI2K4X_Negative(eps:=Main.M46.stEPSBackwardEnable);
EPS_LI2K4X_Negative.setBit(nBits := 0, bValue:= Main.M45.stAxisStatus.fActPosition < 82 OR Main.M46.stAxisStatus.fActPosition > -0.314);



//LI2K4 sequenct move : OUT->IN Y move first and then X moves IN->OUT X moves first then Y

(*fbLI2K4States(
    stMotionStage1:=Main.M45,
    stMotionStage2:=Main.M46,
    astPositionState1:=aLI2K4YStates,
    astPositionState2:=aLI2K4XStates,
    eEnumSet:=li2k4_enumSet,
    eEnumGet:=li2k4_enumGet,
    sDeviceName := 'LI2K4:IP1',
    sTransitionKey := 'LI2K4:IP1-TRANSITION',
    fbFFHWO:=fbFastFaultOutput1,
    fbArbiter:=fbArbiter,
    bEnableMotion:=TRUE,
    bEnableBeamParams:=TRUE,
    bEnablePositionLimits:=TRUE,
);*)
anStateSequenceOrderLI2K4Y[ENUM_LaserCoupling_States.Out] := 2;
anStateSequenceOrderLI2K4Y[ENUM_LaserCoupling_States.Mirror1] := 1;
anStateSequenceOrderLI2K4X[ENUM_LaserCoupling_States.Out] := 1;
anStateSequenceOrderLI2K4X[ENUM_LaserCoupling_States.Mirror1] := 2;

fbFastFault(
    i_xOK:=li2k4_enumGet<>0,
    i_xAutoReset:=TRUE,
    i_DevName:='LI2K4:IP1',
    i_Desc:='LI2K4 is in a transition state.',
    i_TypeCode:=16#1005,
    io_fbFFHWO:=fbFastFaultOutput1
);

fbLI2K4States(
    bReset:=bLI2K4StatesReset,
    anStateSequenceOrder1:=anStateSequenceOrderLI2K4Y,
    anStateSequenceOrder2:=anStateSequenceOrderLI2K4X,
    fbPositionState1D1:=fbLI2K4YStates,
    fbPositionState1D2:=fbLI2K4XStates,
    stMotionStage1:=Main.M45,
    stMotionStage2:=Main.M46,
    astPositionState1:=aLI2K4YStates,
    astPositionState2:=aLI2K4XStates,
    eEnumSet:=li2k4_enumSet,
    eEnumGet:=li2k4_enumGet,
    sDeviceName := 'LI2K4:IP1',
    sTransitionKey := 'LI2K4:IP1-TRANSITION',
    fbFFHWO:=fbFastFaultOutput1,
    fbArbiter:=fbArbiter,
    bEnableMotion:=TRUE,
    bEnableBeamParams:=TRUE,
    bEnablePositionLimits:=TRUE,
);

END_PROGRAM

// ---- POUs/Sequence_Mover/FB_SequenceMover2D.TcPOU
FUNCTION_BLOCK FB_SequenceMover2D
VAR_IN_OUT
    // Set this to a nonzero value to request a new move. It will be reset to zero every cycle. This should be hooked up to a user's EPICS enum input.
    eEnumSet: UINT;
    // The current state index, or zero if we are not at a state. This should be hooked up to a user's EPICS enum output.
    eEnumGet: UINT;
    // The fast fault output to fault to.
    fbFFHWO: FB_HardwareFFOutput;
    // The arbiter to request beam conditions from.
    fbArbiter: FB_Arbiter;

    // The motor to move.
    stMotionStage1: ST_MotionStage;
    // All possible position states, including unused/invalid states.
    {attribute 'pytmc' := '
        pv: STATE:M1
        io: io
        expand: :%.2d
    '}
    astPositionState1: ARRAY[1..GeneralConstants.MAX_STATES] OF ST_PositionState;
    // The motor to move.
    stMotionStage2: ST_MotionStage;
    // All possible position states, including unused/invalid states.
    {attribute 'pytmc' := '
        pv: STATE:M2
        io: io
        expand: :%.2d
    '}
    astPositionState2: ARRAY[1..GeneralConstants.MAX_STATES] OF ST_PositionState;

    fbPositionState1D1 : FB_PositionStatePMPS1D;
    fbPositionState1D2 : FB_PositionStatePMPS1D;


END_VAR
VAR_INPUT
    bReset : BOOL;

    // Index is state enum value. Value at index is sequence order for that state as a goal for the specified axis number.
    // e.g. if state number 2 needs axis 1 to move second, then in index 2 put a 2 for axis 1 and for index 2 on axis 2 put a 1.
    anStateSequenceOrder1 : ARRAY[1...GeneralConstants.MAX_STATES] OF UINT;
    anStateSequenceOrder2 : ARRAY[1...GeneralConstants.MAX_STATES] OF UINT;

    // Set this to TRUE to enable input state moves, or FALSE to disable them.
    bEnableMotion: BOOL;
    // Set this to TRUE to enable beam parameter checks, or FALSE to disable them.
    bEnableBeamParams: BOOL;
    // Set this to TRUE to enable position limit checks, or FALSE to disable them.
    bEnablePositionLimits: BOOL;
    // The name of the device for use in the PMPS DB lookup and diagnostic screens.
    sDeviceName: STRING;
    // The name of the transition state in the PMPS database.
    sTransitionKey: STRING;
 (*   // Normal EPICS inputs, gathered into a single struct
    {attribute 'pytmc' := 'pv: STATE'}
    stEpicsToPlc: ST_StateEpicsToPlc;
    // PMPS EPICS inputs, gathered into a single struct
    {attribute 'pytmc' := 'pv: STATE'}
    stPMPSEpicsToPlc: ST_StatePMPSEpicsToPlc;
*)
    // Set this to TRUE to re-read the loaded database immediately (useful for debug)
     bReadDBNow: BOOL;
END_VAR
VAR_OUTPUT
    // Normal EPICS outputs, gathered into a single struct
    {attribute 'pytmc' := 'pv: STATE'}
    stPlcToEpics: ST_StatePlcToEpics;
    // PMPS EPICS outputs, gathered into a single struct
    {attribute 'pytmc' := 'pv: STATE'}
    stPMPSPlcToEpics: ST_StatePMPSPlcToEpics;
    // The PMPS database lookup associated with the current position state.
    stDbStateParams: ST_DbStateParams;
END_VAR
VAR
    tonStateSequenceTimeout : TON;
    tStateSequenceTimeoutTime : TIME := T#5s;
    nGoal: UINT;
    nState: UINT;
    // The current state index of the 1st axis state mover
    eEnumGet1: UINT;
    // The current state index of the 2nd axis state mover
    eEnumGet2: UINT;
     // Normal EPICS inputs, gathered into a single struct
    {attribute 'pytmc' := 'pv: STATE'}
    stEpicsToPlc: ST_StateEpicsToPlc;
    // PMPS EPICS inputs, gathered into a single struct
    {attribute 'pytmc' := 'pv: STATE'}
    stPMPSEpicsToPlc: ST_StatePMPSEpicsToPlc;
END_VAR


IF bReset THEN
    bReset := FALSE;
    nState := 0;
END_IF

CASE nState OF
    0:
        IF eEnumSet <> 0 THEN
            nGoal := eEnumSet;
            nState := nState + 1;
        ELSE
            fbPositionState1D1(
                stMotionStage:=stMotionStage1,
                astPositionState:=astPositionState1,
                eEnumSet:=eEnumSet,
                eEnumGet:=eEnumGet1,
                sDeviceName:=sDeviceName,
                sTransitionKey:=sTransitionKey,
                fbFFHWO:=fbFFHWO,
                fbArbiter:=fbArbiter,
                bEnableMotion:=bEnableMotion,
                bEnableBeamParams:=bEnableBeamParams,
                bEnablePositionLimits:=bEnablePositionLimits,
                stEpicsToPlc:=stEpicsToPlc,
                stPMPSEpicsToPlc:=stPMPSEpicsToPlc,
                stDbStateParams=>stDbStateParams,
                stPlcToEpics=>stPlcToEpics,
                stPMPSPlcToEpics=>stPMPSPlcToEpics,
            );
            fbPositionState1D2(
                stMotionStage:=stMotionStage2,
                astPositionState:=astPositionState2,
                eEnumSet:=eEnumSet,
                eEnumGet:=eEnumGet2,
                sDeviceName:=sDeviceName,
                sTransitionKey:=sTransitionKey,
                fbFFHWO:=fbFFHWO,
                fbArbiter:=fbArbiter,
                bEnableMotion:=bEnableMotion,
                bEnableBeamParams:=bEnableBeamParams,
                bEnablePositionLimits:=bEnablePositionLimits,
                stEpicsToPlc:=stEpicsToPlc,
                stPMPSEpicsToPlc:=stPMPSEpicsToPlc,
                stDbStateParams=>stDbStateParams,
                stPlcToEpics=>stPlcToEpics,
                stPMPSPlcToEpics=>stPMPSPlcToEpics,
            );
        END_IF
        tonStateSequenceTimeout(IN:=FALSE);
    1:
        IF anStateSequenceOrder1[nGoal] <= anStateSequenceOrder2[nGoal] THEN
            // Move 1 then 2
            fbPositionState1D1(
                stMotionStage:=stMotionStage1,
                astPositionState:=astPositionState1,
                eEnumSet:=eEnumSet,
                eEnumGet:=eEnumGet1,
                sDeviceName:=sDeviceName,
                sTransitionKey:=sTransitionKey,
                fbFFHWO:=fbFFHWO,
                fbArbiter:=fbArbiter,
                bEnableMotion:=bEnableMotion,
                bEnableBeamParams:=bEnableBeamParams,
                bEnablePositionLimits:=bEnablePositionLimits,
                stEpicsToPlc:=stEpicsToPlc,
                stPMPSEpicsToPlc:=stPMPSEpicsToPlc,
                stDbStateParams=>stDbStateParams,
                stPlcToEpics=>stPlcToEpics,
                stPMPSPlcToEpics=>stPMPSPlcToEpics,
            );
            tonStateSequenceTimeout(IN:=NOT stMotionStage1.bBusy,PT:=tStateSequenceTimeoutTime);
            IF stMotionStage1.Axis.NcToPlc.ActPos >= astPositionState1[nGoal].fPosition - astPositionState1[nGoal].fDelta AND
                stMotionStage1.Axis.NcToPlc.ActPos <= astPositionState1[nGoal].fPosition + astPositionState1[nGoal].fDelta THEN
                eEnumGet1 := nGoal;
                eEnumSet := nGoal;
                tonStateSequenceTimeout(IN:=FALSE);
                nState := 10;
            ELSIF tonStateSequenceTimeout.Q THEN
                nState := 0;
            END_IF
        ELSIF anStateSequenceOrder1[nGoal] > anStateSequenceOrder2[nGoal] THEN
            // Move 2 then 1
            fbPositionState1D2(
                stMotionStage:=stMotionStage2,
                astPositionState:=astPositionState2,
                eEnumSet:=eEnumSet,
                eEnumGet:=eEnumGet2,
                sDeviceName:=sDeviceName,
                sTransitionKey:=sTransitionKey,
                fbFFHWO:=fbFFHWO,
                fbArbiter:=fbArbiter,
                bEnableMotion:=bEnableMotion,
                bEnableBeamParams:=bEnableBeamParams,
                bEnablePositionLimits:=bEnablePositionLimits,
                stEpicsToPlc:=stEpicsToPlc,
                stPMPSEpicsToPlc:=stPMPSEpicsToPlc,
                stDbStateParams=>stDbStateParams,
                stPlcToEpics=>stPlcToEpics,
                stPMPSPlcToEpics=>stPMPSPlcToEpics,
            );
            tonStateSequenceTimeout(IN:=NOT stMotionStage2.bBusy,PT:=tStateSequenceTimeoutTime);
            IF stMotionStage2.Axis.NcToPlc.ActPos >= astPositionState2[nGoal].fPosition - astPositionState2[nGoal].fDelta AND
                stMotionStage2.Axis.NcToPlc.ActPos <= astPositionState2[nGoal].fPosition + astPositionState2[nGoal].fDelta THEN
                eEnumGet2 := nGoal;
                eEnumSet := nGoal;
                tonStateSequenceTimeout(IN:=FALSE);
                nState := 20;
            ELSIF tonStateSequenceTimeout.Q THEN
                nState := 0;
            END_IF
        END_IF
    10: // Move 2 after 1
        fbPositionState1D2(
            stMotionStage:=stMotionStage2,
            astPositionState:=astPositionState2,
            eEnumSet:=eEnumSet,
            eEnumGet:=eEnumGet2,
            sDeviceName:=sDeviceName,
            sTransitionKey:=sTransitionKey,
            fbFFHWO:=fbFFHWO,
            fbArbiter:=fbArbiter,
            bEnableMotion:=bEnableMotion,
            bEnableBeamParams:=bEnableBeamParams,
            bEnablePositionLimits:=bEnablePositionLimits,
            stEpicsToPlc:=stEpicsToPlc,
            stPMPSEpicsToPlc:=stPMPSEpicsToPlc,
            stDbStateParams=>stDbStateParams,
            stPlcToEpics=>stPlcToEpics,
            stPMPSPlcToEpics=>stPMPSPlcToEpics,
        );
        tonStateSequenceTimeout(IN:=NOT stMotionStage2.bBusy,PT:=tStateSequenceTimeoutTime);
        IF stMotionStage2.Axis.NcToPlc.ActPos >= astPositionState2[nGoal].fPosition - astPositionState2[nGoal].fDelta AND
            stMotionStage2.Axis.NcToPlc.ActPos <= astPositionState2[nGoal].fPosition + astPositionState2[nGoal].fDelta THEN
            eEnumGet2 := nGoal;
            nState := 0;
            tonStateSequenceTimeout(IN:=FALSE);
        ELSIF tonStateSequenceTimeout.Q THEN
            nState := 0;
        END_IF
    20: // Move 1 after 2
        fbPositionState1D1(
            stMotionStage:=stMotionStage1,
            astPositionState:=astPositionState1,
            eEnumSet:=eEnumSet,
            eEnumGet:=eEnumGet1,
            sDeviceName:=sDeviceName,
            sTransitionKey:=sTransitionKey,
            fbFFHWO:=fbFFHWO,
            fbArbiter:=fbArbiter,
            bEnableMotion:=bEnableMotion,
            bEnableBeamParams:=bEnableBeamParams,
            bEnablePositionLimits:=bEnablePositionLimits,
            stEpicsToPlc:=stEpicsToPlc,
            stPMPSEpicsToPlc:=stPMPSEpicsToPlc,
            stDbStateParams=>stDbStateParams,
            stPlcToEpics=>stPlcToEpics,
            stPMPSPlcToEpics=>stPMPSPlcToEpics,
        );
        tonStateSequenceTimeout(IN:=NOT stMotionStage1.bBusy,PT:=tStateSequenceTimeoutTime);
        IF stMotionStage1.Axis.NcToPlc.ActPos >= astPositionState1[nGoal].fPosition - astPositionState1[nGoal].fDelta AND
            stMotionStage1.Axis.NcToPlc.ActPos <= astPositionState1[nGoal].fPosition + astPositionState1[nGoal].fDelta THEN
            eEnumGet1 := nGoal;
            nState := 0;
            tonStateSequenceTimeout(IN:=FALSE);
        ELSIF tonStateSequenceTimeout.Q THEN
            nState := 0;
        END_IF
END_CASE

IF eEnumGet1 = eEnumGet2 THEN
    eEnumGet := eEnumGet1;
ELSE
    eEnumGet := 0;
END_IF
stEpicsToPlc.bReset := FALSE;

END_FUNCTION_BLOCK

// ---- POUs/PRG_PA1K4_PF.TcPOU
PROGRAM PRG_PA1K4_PF
VAR
    fbMotionPA1K4: FB_MotionStage;{attribute 'pytmc' := '
        pv: PA1K4:PF
        io: io
    '}
    fbPA1K4States: FB_PositionStatePMPS1D;
    {attribute 'pytmc' := '
        pv: PA1K4:PF:STATE:SET
        io: io
    '}
    pa1k4_enumSet: ENUM_Sample_Calibration_States;
     {attribute 'pytmc' := '
        pv: PA1K4:PF:STATE:GET
        io: i
    '}
    pa1k4_enumGet: ENUM_Sample_Calibration_States;
    fbStateSetup: FB_StateSetupHelper;
    stDefault: ST_PositionState :=(
        fDelta :=2.0,
        fVelocity := 5.0,
        bMoveOk := TRUE,
        bValid := TRUE
    );
    aPA1K4States: ARRAY[1..GeneralConstants.MAX_STATES] OF ST_PositionState;



END_VAR

fbMotionPA1K4(stMotionStage:=Main.M47);

fbStateSetup(stPositionState:=stDefault, bSetDefault:=TRUE);
fbStateSetup(stPositionState:=aPA1K4States[ENUM_Sample_Calibration_States.OUT],fdelta := 2.0, sName := 'OUT', fPosition:=180.0);
fbStateSetup(stPositionState:=aPA1K4States[ENUM_Sample_Calibration_States.Target1], fdelta := 2.0, sName := 'TARGET1', fPosition:=160.0);
fbStateSetup(stPositionState:=aPA1K4States[ENUM_Sample_Calibration_States.Target2], fdelta := 2.0, sName := 'TARGET2', fPosition:=140.0);
fbStateSetup(stPositionState:=aPA1K4States[ENUM_Sample_Calibration_States.Target3], fdelta := 2.0, sName := 'TARGET3', fPosition:=121.0);
fbStateSetup(stPositionState:=aPA1K4States[ENUM_Sample_Calibration_States.Target4], fdelta := 2.0, sName := 'TARGET4', fPosition:=101.0);
fbStateSetup(stPositionState:=aPA1K4States[ENUM_Sample_Calibration_States.Target5], fdelta := 2.0, sName := 'TARGET5', fPosition:=81.0);
//target 6 and 7 because is recoered on 7-31-25, those were hided on 05-13-25
fbStateSetup(stPositionState:=aPA1K4States[ENUM_Sample_Calibration_States.Target6], fdelta := 2.0, sName := 'TARGET6', fPosition:=61.0);
fbStateSetup(stPositionState:=aPA1K4States[ENUM_Sample_Calibration_States.Target7], fdelta := 2.0, sName := 'TARGET7', fPosition:=41.0);
//PMPS
aPA1K4States[ENUM_Sample_Calibration_States.OUT].stPMPS.sPmpsState := 'PA1K4:PF-OUT';
aPA1K4States[ENUM_Sample_Calibration_States.Target1].stPMPS.sPmpsState := 'PA1K4:PF-TARGET1';
aPA1K4States[ENUM_Sample_Calibration_States.Target2].stPMPS.sPmpsState := 'PA1K4:PF-TARGET2';
aPA1K4States[ENUM_Sample_Calibration_States.Target3].stPMPS.sPmpsState := 'PA1K4:PF-TARGET3';
aPA1K4States[ENUM_Sample_Calibration_States.Target4].stPMPS.sPmpsState := 'PA1K4:PF-TARGET4';
aPA1K4States[ENUM_Sample_Calibration_States.Target5].stPMPS.sPmpsState := 'PA1K4:PF-TARGET5';
//hide target 6 and 7 because it cannot fully reached 5-13-25 and targets are recovered 7-31-25
aPA1K4States[ENUM_Sample_Calibration_States.Target6].stPMPS.sPmpsState := 'PA1K4:PF-TARGET6';
aPA1K4States[ENUM_Sample_Calibration_States.Target7].stPMPS.sPmpsState := 'PA1K4:PF-TARGET7';


fbPA1K4States(
    stMotionStage:=Main.M47,
    astPositionState:=aPA1K4States,
    eEnumSet:=pa1k4_enumSet,
    eEnumGet:=pa1k4_enumGet,
    sDeviceName := 'PA1K4:PF',
    sTransitionKey := 'PA1K4:PF-TRANSITION',
    fbFFHWO:=fbFastFaultOutput1,
    fbArbiter:=fbArbiter,
    bEnableMotion:=TRUE,
    bEnableBeamParams:=TRUE,
    bEnablePositionLimits:=TRUE,
);

END_PROGRAM

// ---- POUs/PRG_3_PMPS_POST.TcPOU
PROGRAM PRG_3_PMPS_POST
VAR
    fbArbiterIO: FB_SubSysToArbiter_IO;
    fb_vetoArbiter: FB_VetoArbiter;

    bST3K4_Veto: BOOL;
    bST1K4_Veto: BOOL;
    bM1K1Veto: BOOL;
    bM1K3Veto: BOOL;
    bST4K4_Veto:BOOL;
END_VAR

bST3K4_Veto := PMPS_GVL.stCurrentBeamParameters.aVetoDevices[PMPS.K_Stopper.ST3K4];
bST1K4_Veto := PMPS_GVL.stCurrentBeamParameters.aVetoDevices[PMPS.K_Stopper.ST1K4];
bST4K4_Veto := PMPS_GVL.stCurrentBeamParameters.aVetoDevices[PMPS.K_Stopper.ST4K4];
bM1K1Veto := NOT PMPS_GVL.stCurrentBeamParameters.aVetoDevices[PMPS.K_Stopper.MR1K1_OUT]
                AND PMPS_GVL.stCurrentBeamParameters.aVetoDevices[PMPS.K_Stopper.MR1K1_IN];
bM1K3Veto := NOT PMPS_GVL.stCurrentBeamParameters.aVetoDevices[PMPS.K_Stopper.MR1K3_OUT]
                AND PMPS_GVL.stCurrentBeamParameters.aVetoDevices[PMPS.K_Stopper.MR1K3_IN];


fbArbiterIO(
    i_bVeto:=bST3K4_Veto OR bM1K1Veto OR bST1K4_Veto,
    Arbiter:=fbArbiter,
    fbFFHWO:=fbFastFaultOutput1);

fb_vetoArbiter(bVeto:=bST4K4_Veto OR bST3K4_Veto OR bST1K4_Veto OR bM1K1Veto OR bM1K3Veto,
                HigherAuthority := GVL_PMPS.fbArbiter,
                LowerAuthority := GVL_PMPS.fbArbiter2,
                FFO := GVL_PMPS.fbFastFaultOutput2);

fbFastFaultOutput1.Execute(i_xVeto:=bST3K4_Veto OR bST1K4_Veto OR bM1K1Veto OR bM1K3Veto);
fbFastFaultOutput2.Execute(i_xVeto:=bST3K4_Veto OR bST1K4_Veto OR bM1K1Veto OR bST4K4_Veto OR bM1K3Veto); // Adding TXI MR1K3 veto in

END_PROGRAM

// ---- POUs/PRG_ST5K4_TMO_TERM_FIXED.TcPOU
PROGRAM PRG_ST5K4_TMO_TERM_FIXED
VAR
    {attribute 'pytmc' := 'pv: ST5K4:TMO_TERM_FIXED'}
    {attribute 'TcLinkTo' := 	'.i_xInsertedLS	:=	TIIB[ST4K4-EP2338]^Channel 4^Input;
                                 .i_xRetractedLS:=	TIIB[ST4K4-EP2338]^Channel 3^Input;
                                 .q_xInsert_DO	:=	TIIB[ST4K4-EP2338]^Channel 9^Output
    '}
    ST4K4: FB_MotionPneumaticActuator;
    ibPMPS_OK : BOOL;
END_VAR

ST4K4(
    ibInsertOK:= TRUE,
    ibRetractOK:= TRUE,
    ibPMPS_OK:= ibPMPS_OK,
    ibSingleCntrl:= TRUE ,
    ibCntrlHold:= TRUE,
    ibOverrideInterlock:= ,
    i_xReset:= ,
    stPneumaticActuator=> ,
    xMPS_OK=>  ,
    io_fbFFHWO:= fbFastFaultOutput2  ); // Do Stoppers send MPS signal?

END_PROGRAM

// ---- POUs/temp/FB_SLITS_POWER.TcPOU
FUNCTION_BLOCK FB_SLITS_POWER EXTENDS FB_SLITS
VAR_INPUT
END_VAR
VAR
     {attribute 'pytmc' := '
        pv: FSW
    '}
    fbFlowSwitch: FB_XTES_Flowswitch;


    //RTDs
    {attribute 'pytmc' := '
        pv: TOP:RTD:01
    '}
    RTD_TOP_1: FB_TempSensor;
    {attribute 'pytmc' := '
        pv: TOP:RTD:02
    '}
    RTD_TOP_2: FB_TempSensor;
    {attribute 'pytmc' := '
        pv: BOTTOM:RTD:01
    '}
    RTD_Bottom_1: FB_TempSensor;
    {attribute 'pytmc' := '
        pv: BOTTOM:RTD:02
    '}
    RTD_Bottom_2: FB_TempSensor;

    {attribute 'pytmc' := '
        pv: NORTH:RTD:01
    '}
    RTD_North_1: FB_TempSensor;
    {attribute 'pytmc' := '
        pv: NORTH:RTD:02
    '}
    RTD_North_2: FB_TempSensor;
    {attribute 'pytmc' := '
        pv: SOUTH:RTD:01
    '}
    RTD_South_1: FB_TempSensor;
    {attribute 'pytmc' := '
        pv: SOUTH:RTD:02
    '}
    RTD_South_2: FB_TempSensor;


END_VAR


ACT_RTDs();

ACTION ACT_RTDs:
////RTDs
RTD_TOP_1();
RTD_TOP_2();
RTD_Bottom_1();
RTD_Bottom_2();
RTD_North_1();
RTD_North_2();
RTD_South_1();
RTD_South_2();

//Flow Switch
fbFlowSwitch();
END_ACTION

END_FUNCTION_BLOCK

// ---- POUs/temp/FB_SLITS_SCATTER.TcPOU
FUNCTION_BLOCK FB_SLITS_SCATTER EXTENDS FB_SLITS
VAR_INPUT
END_VAR
VAR
    


END_VAR

END_FUNCTION_BLOCK

// ---- POUs/temp/PRG_SL2K4_SCATTER.TcPOU
PROGRAM PRG_SL2K4_SCATTER
VAR
    {attribute 'pytmc' := '
        pv: SL2K4:SCATTER
        io: io
    '}
    fbSL2K4: FB_SLITS;
    //GET PMPS Move Ok bit
    // Default True until it is properly linked to PMPS bit
    bMoveOk:BOOL :=TRUE;
    {attribute 'pytmc' := '
    pv: SL2K4:SCATTER:GO;
    io: io;
    field: ZNAM False;
    field: ONAM True;
    '}
    bExecuteMotion :BOOL :=FALSE;
    bTest:BOOL:=FALSE;
    //for testing purposes only. comment-out/delete once done.
    mcPower : ARRAY [1..4] OF MC_POWER;


    (*Offsets*)
    (* Absolute encoder value at the HLS + Absolure eoncoder value at the centered beam *)
    rEncoderOffsetTop: REAL := -15; (* 0+(-15)*)
    rEncoderOffsetBottom: REAL := -15; (* 0+(-15)*)
    rEncoderOffsetNorth: REAL := -15;(* 0+(-15)*)
    rEncoderOffsetSouth: REAL := -15;(* 0+(-15)*)

END_VAR



fbSL2K4.bMoveOk := bMoveOk;

//for testing purposes only. comment-out/delete once done.
If (bTest) THEN
mcPower[1](axis:=Main.M23.Axis, Enable:=bTest, enable_positive:=Main.M23.bLimitForwardEnable, enable_negative:=Main.M23.bLimitBackwardEnable);
mcPower[2](axis:=Main.M24.Axis, Enable:=bTest, enable_positive:=Main.M24.bLimitForwardEnable, enable_negative:=Main.M24.bLimitBackwardEnable);
mcPower[3](axis:=Main.M25.Axis, Enable:=bTest, enable_positive:=Main.M25.bLimitForwardEnable, enable_negative:=Main.M25.bLimitBackwardEnable);
mcPower[4](axis:=Main.M26.Axis, Enable:=bTest, enable_positive:=Main.M26.bLimitForwardEnable, enable_negative:=Main.M26.bLimitBackwardEnable);
ELSE

//Homing routine parameters
Main.M24.fHomePosition:= 0;
Main.M23.fHomePosition:= -30.6;
Main.M25.fHomePosition:= 0;
Main.M26.fHomePosition:= -30.51;

Main.M24.nHomingMode := ENUM_EpicsHomeCmd.HIGH_LIMIT;
Main.M23.nHomingMode := ENUM_EpicsHomeCmd.LOW_LIMIT;
Main.M25.nHomingMode := ENUM_EpicsHomeCmd.HIGH_LIMIT;
Main.M26.nHomingMode := ENUM_EpicsHomeCmd.LOW_LIMIT;


fbSL2K4.rEncoderOffsetTop := rEncoderOffsetTop;
fbSL2K4.rEncoderOffsetBottom := rEncoderOffsetBottom;
fbSL2K4.rEncoderOffsetNorth := rEncoderOffsetNorth;
fbSL2K4.rEncoderOffsetSouth := rEncoderOffsetSouth;

fbSL2K4(stTopBlade:=  Main.M24,
        stBottomBlade:= Main.M23,
        stNorthBlade:=  Main.M25,
        stSouthBlade:=  Main.M26,
        bExecuteMotion:=bExecuteMotion,
        io_fbFFHWO := GVL_PMPS.fbFastFaultOutput2,
        fbArbiter := GVL_PMPS.fbArbiter);

//fbSL2K4.M_CheckPMPS(2);



END_IF

END_PROGRAM
